// TwinCAT 3 PLC project Monica
// ProgramVersion: 3.1.4024.12
// libraries:
//   Tc2_Standard, * (Beckhoff Automation GmbH)
//   Tc2_System, * (Beckhoff Automation GmbH)
//   Tc2_Utilities, * (Beckhoff Automation GmbH)
//   Tc3_Module, * (Beckhoff Automation GmbH)
// project tree:
//   DUTs/BF_IDM25/ enBN_IDM_error.TcDUT, stBN_IDM_header_in.TcDUT, stBN_IDM_header_out.TcDUT, stBN_IDM.TcDUT, unBN_IDM_header_in.TcDUT, unBN_IDM_header_out.TcDUT
//   DUTs/ enAccessLevel.TcDUT, enState.TcDUT, structAlarm.TcDUT, structButton.TcDUT, stUserID.TcDUT
//   GVLs/ AXIS.TcGVL, CONST.TcGVL, GVL.TcGVL, HMI.TcGVL, IN.TcGVL, OUT.TcGVL, PERS.TcGVL
//   / PlcTask.TcTTO
//   POUs/05_DRIVER/ FB_BF_IDM25_FULL.TcPOU, FB_BF_IDM25_SIMPLE.TcPOU
//   POUs/10_HMI/FB%27s/ FB_BUTTON.TcPOU (not stored)
//   POUs/10_HMI/ _14_STATE.TcPOU
//   POUs/20_AUTO/FB%27s/ FB_ID_list_man.TcPOU (not stored)
//   POUs/ MAIN.TcPOU
// real-time tasks:
//   TASK PlcTask: cycle T#10ms, priority 20, ADS port 350
// I/O:
//   DEVICE Device 5 (NOV-DP-RAM)
//   DEVICE Device 4 (USB)
//     Box 1 (CX2100 Power Supply)
//   DEVICE Device 1 (EtherCAT), AmsNetId 192.168.20.200.2.1
//     Term 1 (EK1200) [EK1200-5000 EtherCAT Power supply (2A E-Bus)]
//       Term 2 (EL6070-0033) [EL6070-0033 1Ch. Licence key terminal, individual licences]
//       Term 3 (EL1008) [EL1008 8Ch. Dig. Input 24V, 3ms]
//       Term 5 (EL2008) [EL2008 8Ch. Dig. Output 24V, 0.5A]
//       Term 6 (EK1110) [EK1110 EtherCAT extension]
//     Box 7 (EP6228-3032) [EP6228-3032 (IO Link Master Class B)]
//       modules: Module 1 (DeviceState Inputs Device), Module 2 (DeviceState Inputs), Module 3 (IO-Link Slave), Module 4 (empty), Module 5 (IO-Link Slave), Module 6 (empty), Module 7 (empty), Module 8 (empty), Module 9 (empty), Module 10 (empty)
// variable links:
//   Monica/Monica Instance <-> Device 1 (EtherCAT)/Box 7 (EP6228-3032)
//     PlcTask Inputs/GVL.rfid.I_RFID_arr_data <-> Module 3 (IO-Link Slave)/IO-Link Port1_in/Byte 1
//     PlcTask Inputs/GVL.rfid.I_RFID_arr_data @bit {8..56 step 8} <-> Module 3 (IO-Link Slave)/IO-Link Port1_in/Byte {2..8}  (7 links)
//     PlcTask Inputs/GVL.rfid.I_RFID_bitheader1/raw <-> Module 3 (IO-Link Slave)/IO-Link Port1_in/Bitheader 1
//     PlcTask Inputs/GVL.rfid.I_RFID_bitheader2/raw <-> Module 3 (IO-Link Slave)/IO-Link Port1_in/Bitheader 2
//     PlcTask Outputs/GVL.rfid.O_RFID_arr_data <-> Module 3 (IO-Link Slave)/IO-Link Port1_out/Byte 1
//     PlcTask Outputs/GVL.rfid.O_RFID_arr_data @bit {8..56 step 8} <-> Module 3 (IO-Link Slave)/IO-Link Port1_out/Byte {2..8}  (7 links)
//     PlcTask Outputs/GVL.rfid.O_RFID_bitheader/raw <-> Module 3 (IO-Link Slave)/IO-Link Port1_out/Bitheader 1
//     PlcTask Outputs/GVL.rfid.O_RFID_bitheader/raw <-> Module 3 (IO-Link Slave)/IO-Link Port1_out/Bitheader 2

CONFIGURATION Monica
    RESOURCE PLC ON TwinCAT3
        TASK PlcTask(INTERVAL := T#10ms, PRIORITY := 20);
        PROGRAM MAIN WITH PlcTask : MAIN;
    END_RESOURCE
END_CONFIGURATION

// ---- DUTs/BF_IDM25/enBN_IDM_error.TcDUT
{attribute 'qualified_only'}
{attribute 'strict'}
TYPE enBN_IDM_error :
(
	no_error,
	header_missmatch,
	no_power,
	head_failure,
	max_
);
END_TYPE

// ---- DUTs/BF_IDM25/stBN_IDM_header_in.TcDUT
TYPE stBN_IDM_header_in :
STRUCT
	CP	: BIT;  // Codetag Present
	AE	: BIT;  // Job end
	AA	: BIT;  // Job accepted
	AF	: BIT;  // Job error
	zz	: BIT;	// NOT USED
	TB	: BIT;  // Replace TO, Toggle bit
	HF	: BIT;  // Head Failure
	BB	: BIT;	// Power
END_STRUCT
END_TYPE

// ---- DUTs/BF_IDM25/stBN_IDM_header_out.TcDUT
TYPE stBN_IDM_header_out :
STRUCT
	zz	: BIT;		// UNUSED
	AV	: BIT;		// Job, 1 = New job pending
	zy	: BIT;		// UNUSED	   
	GR	: BIT;		// Basic state, 1 = Sofware reset
	zx	: BIT;		// UNUSED	
	zw	: BIT;		// UNUSED	
	KA	: BIT;		// Head on/off, 1 = Head off
	TI	: BIT;		// Toggle bit, 1 = PLC ready to receive next data
	zv	: BIT;		// UNUSED
END_STRUCT
END_TYPE

// ---- DUTs/BF_IDM25/stBN_IDM.TcDUT
TYPE stBN_IDM :
STRUCT
		I_RFID_bitheader1	AT %I*	: unBN_IDM_header_in;		// Bit header for the RFID reader
		I_RFID_bitheader2	AT %I*	: unBN_IDM_header_in;		// Bit header for the RFID reader, must be equal to bitheader1
		I_RFID_arr_data		AT %I*	: ARRAY [0..7] OF BYTE;	// Data array of the RFID reader
		
		O_RFID_bitheader	AT %Q*	: unBN_IDM_header_out;					// output bitfield header for the RFID reader. Link this value to the 2 headers
		O_RFID_arr_data		AT %Q*	: ARRAY [0..7] OF BYTE;	// Data array of the RFID reader
END_STRUCT
END_TYPE

// ---- DUTs/BF_IDM25/unBN_IDM_header_in.TcDUT
TYPE unBN_IDM_header_in :
UNION
	bits	: stBN_IDM_header_in;	// bit access
	raw		: BYTE;				// byte access
END_UNION
END_TYPE

// ---- DUTs/BF_IDM25/unBN_IDM_header_out.TcDUT
TYPE unBN_IDM_header_out :
STRUCT
	bits	: stBN_IDM_header_out;	// bit access
	raw		: BYTE;					// raw access
END_STRUCT
END_TYPE

// ---- DUTs/enAccessLevel.TcDUT
{attribute 'qualified_only'}
{attribute 'strict'}
{attribute 'to_string'}
TYPE enAccessLevel :
(
	logged_out,
	operator,
	maintenance,
	admin,
	help_tec,
	max_
);
END_TYPE

// ---- DUTs/enState.TcDUT
TYPE enState :
	//	MACHINE STATE
(
	StateOFF	,		(*0	OFF 		PLC STARTUP, EMERGENCY STOP	*)
	StateAIRon	,		(*1	AIR OK		AIRPRESSURE ON	 	*)
	StateENGIZED,		(*2	ENERGY OK	ENERGY/SECURITY CIRQUIT CLOSED	*)
	StateREF	,		(*3	HOMING		SYSTEM INITIAL RESET (HOMING AXIS ETC) *)
	StateMANU	,		(*4	MANUEL		MANUEL MODE (TEACH AXIS, MANEL MOVEMENT	*)
	StateINIT	,		(*5	INITIALISE	SYSTEM RESET 	*)
	StateREADY	,		(*6	READY		SYSTEM READY TO START	*)
	StateSTOP	,		(*7	STOP		SYSTEM STOPPED	*)
	StateALARM	,		(*8	ALARM		ALARM ACTIV	*)
	StateSTEP	,		(*9	STEP		STEP BY STEP MODE	*)
	StateEND	,		(*10 END		END MODE (FINISH ALL CYCLES	*)
	StateLEER	,		(*11 EMPTY		
NING TILL EMPTY STATE *)
	StateAUTO			(*12 RUN		RUNNING AUTOMATIC MODE	*)
);
END_TYPE

// ---- DUTs/structAlarm.TcDUT
TYPE structAlarm :
STRUCT
	xAlarmIN	:	BOOL;	//Alarm Trigger
	xAlarmOFF	:	BOOL;	//Alarm übersteuert (wird nicht ausgelöst)
	xAlarmSAVE	:	BOOL;	//Alarm gespeichert (muss quittiert werden)
	xAlarmQUIT	:	BOOL;	//Alarm quittieren
	xAlarmOUT	:	BOOL;	//Alarm aktiv
	tAlarmVERZ	:	TIME;	//Alarmverzögerung
	sAlarmText	:	STRING;	//Alarmtext
	bAlarmNr	:	BYTE;	//Zusatztext #
END_STRUCT
END_TYPE

// ---- DUTs/structButton.TcDUT
TYPE structButton :
STRUCT
	button	:	BOOL;	// BUTTON SIGNAL FROM HMI
	disable	:	BOOL;	// FORCE BUTTON INACTIV
	rtrig	:	BOOL;	// RISING EDGE
	ftrig	:	BOOL;	// FALLING EDGE
	press	:	BOOL;	// BUTTON PRESSED
	on		:	BOOL;	// FUNCTION ON (GREEN)
	error	:	BOOL;	// FUNCTION ERROR (RED)
END_STRUCT
END_TYPE

// ---- DUTs/stUserID.TcDUT
TYPE stUserID :
	(* Retain user ID with a tag number *)
STRUCT
	bArrTag		: ARRAY [0..7] OF BYTE;		// tag number
	sName		: STRING;					// user name
	bLevel		: enAccessLevel;			// access level
END_STRUCT
END_TYPE

// ---- GVLs/AXIS.TcGVL
{attribute 'qualified_only'}
(*******************************************************************)
(* ACHSEN KONSTANTEN *)
(*******************************************************************)
VAR_GLOBAL CONSTANT
	//Axis

END_VAR
VAR_GLOBAL
(*******************************************************************)
(* ACHSEN Variablen *)
(*******************************************************************)

END_VAR

(*******************************************************************)
(* ACHSEN Positionen von HMI*)
(*******************************************************************)	
VAR_GLOBAL RETAIN
													
END_VAR

// ---- GVLs/CONST.TcGVL
{attribute 'qualified_only' := ''}
VAR_GLOBAL CONSTANT
(*******************************************************************)
(* Globale KONSTANTEN *)
(*******************************************************************)
END_VAR

// ---- GVLs/GVL.TcGVL
{attribute 'qualified_only'}
VAR_GLOBAL
(*******************************************************************)
(* Allgemeine Globale Variablen *)
(*******************************************************************)

	rfid : stBN_IDM;

END_VAR

// ---- GVLs/HMI.TcGVL
{attribute 'qualified_only'}
VAR_GLOBAL
(*******************************************************************)
(* Globale HMI Variablen *)
(*******************************************************************)
	xFALSE			: 	BOOL := FALSE;	//ALLWAYS FALSE
	xTRUE			: 	BOOL := TRUE;	//ALLWAYS TRUE

//----------------------------------------------------------------------------------
// Access manager
//----------------------------------------------------------------------------------
	bp_add_user	: structButton;
	bp_del_user	: structButton;
	bp_access	: structButton;
	bp_logout	: structButton;
	st_user_in	: stUserID;
	sUser_tag_in	: STRING;	// user tag in a string forrmat
	
END_VAR

// ---- GVLs/IN.TcGVL
{attribute 'qualified_only'}
VAR_GLOBAL
(*******************************************************************)
(* EINGÄNGE *)
(*******************************************************************)
	(* Modul Digital Eingang*)
	//-EL1008#
	I000_reserve	AT %I*		:	BOOL;			// reserve
	I001_reserve	AT %I*		:	BOOL;			// reserve
	I002_reserve	AT %I*		:	BOOL;			// reserve
	I003_reserve	AT %I*		:	BOOL;			// reserve
	I004_reserve	AT %I*		:	BOOL;			// reserve
	I005_reserve	AT %I*		:	BOOL;			// reserve
	I006_reserve	AT %I*		:	BOOL;			// reserve
	I007_reserve	AT %I*		:	BOOL;			// reserve
	
	
END_VAR

// ---- GVLs/OUT.TcGVL
{attribute 'qualified_only'}
VAR_GLOBAL
(*******************************************************************)
(* AUSGÄNGE *)
(*******************************************************************)
	(* Modul1 *)	
	//-EL2008
	Q000_res				AT %QX0.0		:	BOOL;			// reserve
	Q001_res				AT %QX0.1		:	BOOL;			// reserve
	Q002_res				AT %QX0.2		:	BOOL;			// reserve
	Q003_res				AT %QX0.3		:	BOOL;			// reserve
	Q004_res				AT %QX0.4		:	BOOL;			// reserve
	Q005_res				AT %QX0.5		:	BOOL;			// reserve
	Q006_res				AT %QX0.6		:	BOOL;			// reserve
	Q007_res				AT %QX0.7		:	BOOL;			// reserve

END_VAR

// ---- GVLs/PERS.TcGVL
{attribute 'qualified_only'}
VAR_GLOBAL RETAIN
(***********************************************************************************************)
(* COUNTER *)
(***********************************************************************************************)
	//COUNTER 
	udiTotalOK			:	UDINT;		// Total Counter  OK 
	udiTotalNOK			:	UDINT;		// Total Counter  NOK 
	udiTempOK			:	UDINT;		// Temporary Counter  OK 
	udiTempNOK			:	UDINT;		// Temporary Counter  NOK 
	
	//OPERATING HOURS
	udiCountHon			:	UDINT;		// Operating hours SYSTEM POWER ON [h] 
	udiCount6Mon		:	UDINT;		// Operating hours SYSTEM POWER ON [6min (0.1h)] 
	udiCountHauto		:	UDINT;		// Operating hours SYSTEM IN AUTOMATIC MODE [h] 
	udiCount6Mauto		:	UDINT;		// Operating hours SYSTEM IN AUTOMATIC MODE [6min (0.1h)] 
	
	// user level list
	local_user_list	: ARRAY [0..19] OF stUserID;
END_VAR

// ---- POUs/MAIN.TcPOU
PROGRAM MAIN
VAR
	fb_rfid : FB_BF_IDM25_SIMPLE;
	fb_id_list : FB_ID_list_man;
	
	xRFID_new_value	: BOOL;		// Rising edge for the new value
	sUser_tag_out	: STRING;	// user tag in a string forrmat	
	sCurr_access_level	: STRING;		// current access level in a string format
END_VAR


// update HMI var here ...
_14_STATE();



fb_rfid(rfid_hw:=GVL.rfid);

fb_id_list.string_to_tag(HMI.sUser_tag_in, ADR(HMI.st_user_in.bArrTag));

// get information using RFID tag
IF fb_rfid.xNew_val THEN
	HMI.st_user_in.bArrTag := fb_rfid.last_read;
	
	IF fb_id_list.is_user_in_list(ADR(PERS.local_user_list), ADR(HMI.st_user_in)) THEN
		HMI.st_user_in := fb_id_list.get_user_by_tag(HMI.st_user_in.bArrTag);
		fb_id_list.tag_to_string(ADR(HMI.sUser_tag_in), fb_rfid.last_read);
	ELSE
		MEMSET(ADR(HMI.st_user_in), 0, SIZEOF(stUserID));
		fb_id_list.tag_to_string(ADR(HMI.sUser_tag_in), fb_rfid.last_read);
	END_IF
	// Do it here because we reset all data in the else above
	fb_id_list.tag_to_string(ADR(HMI.sUser_tag_in), fb_rfid.last_read);
	
END_IF

fb_id_list(	stUserIn := HMI.st_user_in,
			stArrList := ADR(PERS.local_user_list),
			xAdd := HMI.bp_add_user.rtrig,
			xDel := HMI.bp_del_user.rtrig,
			xAccess := HMI.bp_access.rtrig OR fb_rfid.xNew_val,
			xLogOut := HMI.bp_logout.rtrig,
			tRestore := T#1S,
			tTimeOut := T#1M);
			
// ------------------
// Resolve output HMI
// ------------------
// check if we can resolve an access
IF fb_id_list.xAccess THEN
	IF fb_id_list.is_user_in_list(ADR(PERS.local_user_list), ADR(HMI.st_user_in)) THEN
		HMI.st_user_in := fb_id_list.get_user_by_tag(fb_id_list.stLastUser.bArrTag);
	END_IF
END_IF
	
fb_id_list.tag_to_string(ADR(sUser_tag_out), fb_id_list.stLastUser.bArrTag);
sCurr_access_level := TO_STRING(fb_id_list.iCurrLevel);

END_PROGRAM

// ---- POUs/05_DRIVER/FB_BF_IDM25_SIMPLE.TcPOU
FUNCTION_BLOCK FB_BF_IDM25_SIMPLE
VAR_INPUT
	rfid_hw		: stBN_IDM;
END_VAR
VAR_OUTPUT
	xNew_val	: BOOL;		// New value available
	last_read	: ARRAY [0..7] OF BYTE;		// array of the last RFID values inside the reader
	error		: BOOL;						// To TRUE if the RFID reader is in error
	error_id	: enBN_IDM_error;				// error id
END_VAR
VAR
	i : INT;
	xRt_new_value	: R_TRIG;
END_VAR

error_id := 0;

IF rfid_hw.I_RFID_bitheader1.raw = rfid_hw.I_RFID_bitheader2.raw THEN
	
	IF NOT rfid_hw.I_RFID_bitheader1.bits.BB THEN
		error_id := enBN_IDM_error.no_power;
		
	ELSIF rfid_hw.I_RFID_bitheader1.bits.HF THEN
		error_id := enBN_IDM_error.head_failure;
		
	ELSIF rfid_hw.I_RFID_bitheader1.bits.CP THEN
		MEMCPY(ADR(last_read), ADR(rfid_hw), SIZEOF(last_read));
		
	END_IF
	
ELSE
	error_id := enBN_IDM_error.header_missmatch;
END_IF
xRt_new_value(CLK := rfid_hw.I_RFID_bitheader1.bits.CP);
xNew_val := xRt_new_value.Q;
error := error_id <> enBN_IDM_error.no_error;

END_FUNCTION_BLOCK

// ---- POUs/10_HMI/_14_STATE.TcPOU
PROGRAM _14_STATE
(****************************************************************************)
//STATE PROGRAMM
//	- Control Buttons
//	- Status Anlage
//
//	09.09.2020 / MAD
//
//	Version:			--> Anpassen Projekt 20116
(****************************************************************************)
VAR
	//Control Buttons
	fb_bp_add		: FB_BUTTON;
	fb_bp_del		: FB_BUTTON;
	fb_bp_access	: FB_BUTTON;
	fb_bp_logout	: FB_BUTTON;
END_VAR

//****************************************************************************
// 	CONTROL BUTTONS
//****************************************************************************
//	AUTO 
fb_bp_add(pbtIN:= ADR(HMI.bp_add_user),
	xINdis:= FALSE, 
	xINon:= FALSE, 
	xINerr:= FALSE);

fb_bp_del(pbtIN:= ADR(HMI.bp_del_user),
	xINdis:= FALSE, 
	xINon:= FALSE,
	xINerr:= FALSE);

fb_bp_access(pbtIN:= ADR(HMI.bp_access),
	xINdis:= FALSE, 
	xINon:= FALSE,
	xINerr:= FALSE);

fb_bp_logout(pbtIN:= ADR(HMI.bp_logout),
	xINdis:= FALSE, 
	xINon:= FALSE,
	xINerr:= FALSE);

END_PROGRAM

// ---- POUs/05_DRIVER/FB_BF_IDM25_FULL.TcPOU
FUNCTION_BLOCK FB_BF_IDM25_FULL
VAR_INPUT
END_VAR
VAR_OUTPUT
	xDATA_READY	: BOOL;		// Data are ready and valid in the RFID reader
	xBUSY_READ	: BOOL;		// We are reading values and acknowledging the RFID reader
	xBUSY_WRITE	: BOOL;		// We are writing values and acknowledging the RFID reader
	iRFID_version : WORD;	// RFID version
END_VAR
VAR
	xInit_done	: BOOL;	// TRUE when the initialisation sequence is done (read the devie version)
	xCLK_READ	: BOOL;	// clock signal to ensure BUSY_READ flag is not reset before the task has update itself (manage falling edge)
	xCLK_WRITE	: BOOL;	// clock signal to ensure BUSY_WRITE flag is not reset before the task has update itself (manage falling edge)
END_VAR
VAR_IN_OUT
	rfid_hw		: stBN_IDM;
END_VAR

IF xBUSY_READ AND NOT xCLK_READ THEN
	xBUSY_READ := FALSE;
END_IF
xCLK_READ := xBUSY_READ;

IF xBUSY_WRITE AND NOT xCLK_WRITE THEN
	xBUSY_WRITE := FALSE;
	xCLK_WRITE := TRUE;
END_IF

METHOD FB_init : BOOL
(* Constructor of the FB_init
 *)
VAR_INPUT
	bInitRetains : BOOL; // if TRUE, the retain variables are initialized (warm start / cold start)
	bInCopyCode : BOOL;  // if TRUE, the instance afterwards gets moved into the copy code (online change)
END_VAR
END_METHOD

METHOD PRIVATE read_ack : BOOL
(* Acknoledge the hardware from a valid read
 * return TRUE if rfid hardware is not busy
 *)
VAR_INPUT
END_VAR

VAR
	xRet: BOOL := FALSE;
END_VAR
read_ack:=FALSE;
IF NOT THIS.xBUSY THEN
	THIS.rfid_hw.O_RFID_bitheader1 := 16#01;
	THIS.rfid_hw.O_RFID_bitheader2 := THIS.rfid_hw.O_RFID_bitheader1;
	THIS.xBUSY := TRUE;
	THIS.xCLK := FALSE;
	read_ack:=TRUE;
END_IF
END_METHOD

METHOD PUBLIC read_array : BOOL
(* Read the full array of data from the RFID
 * This function reset the BUSY flag from its parent FB
 *
 * How to use it:
 * When the parent READY flag is set, use this method to read all the values
 * and store them into your local variable
 * IF fb_myFb.xReady THEN
 *     fb_myFb.read(ADR(my_local_array));
  * END_IF
 *)
VAR_INPUT
	pArrData	: POINTER TO ARRAY [0..7] OF BYTE;	// pointer where the data needs to be stored
END_VAR

VAR
	i: INT;
	xRet : BOOL := FALSE; 
END_VAR
read_array := FALSE;
IF THIS.xReady AND NOT THIS.xBUSY THEN
	FOR i:=0 TO 7 BY 1 DO
		^pArrData[i] := THIS.rfid_hw.I_RFID_arr_data[i]; 
	END_FOR
	
	read_array := THIS.read_ack();
END_IF
END_METHOD

METHOD PRIVATE write_reset : BOOL
VAR_INPUT
END_VAR
 THIS.rfid_hw.O_RFID_bitheader1 := BN_IDM_flag_out.BB;
END_METHOD

END_FUNCTION_BLOCK
